// TIA Portal V18 export
DATA_BLOCK "ST10_RecipeActiveDB"   // DB1064
{ S7_Optimized_Access := 'FALSE' }
VERSION : 0.1
// stored: AutoNumber false, DBAccessibleFromOPCUA true, DBAccessibleFromWebserver true, IsOnlyStoredInLoadMemory false, IsWriteProtectedInAS false
   VAR RETAIN
      Recipe : Struct   // System Defined=
         RecipeTag : String[50];   // 配方名称ID
         RecordName : String[50];   // 数据记录名称
         PreConfigType : String[50];   // 待切换数据记录名称
         Pulse : Bool;
         Trigger : Bool;   // 配方切换触发
         PosEdg : Bool;
         Alarm : Bool;
         Ret : Bool;
         Equal : Bool;
         Pls : Bool;
         "time" : Int;
         Spare : Array[0..38] of Byte;
         DataRecord_TransferStatus : Int;   // 数据记录传送状态
      END_STRUCT;
      ParameterElement : Struct
         TypeName : String[50];   // System Defined=
         TypeID : Int;   // System define= product type for parameters of servo ,press and so on
         FixtureID : Array[0..5] of Int;
         FestoAxis : "RecipeAxis";
         PressRgramNo { S7_SetPoint := 'True'} : Array[0..60] of DInt;
         ProcessParameter { S7_SetPoint := 'True'} : "MEStoPLC_RecipeData_OP220";
      END_STRUCT;
   END_VAR
BEGIN
END_DATA_BLOCK
